# B&R Automation Studio project Tmp_Explorer_V1
Automation Studio 4.12.7.113 SP; technology packages: mappView 5.24.4

## Configuration Simulation

CPU PC_any, AutomationRuntime B4.53, Build 4.1.2, Vc V4.52.0

### Task classes (Cpu.sw)
```
Cyclic#8 (cycle 10000 us):
  FileExplor <- mappFileExplorer.FileExplorer.prg
  NETdevice <- mappFileExplorer.NETdevice.prg
  USBdevice <- mappFileExplorer.USBdevice.prg
Binaries: TCData, mvLoader, udbdef, ashwac, Role, ashwd, arconfig, iomap, OpcUaMap, asfw, sysconf, User
Libraries: standard, asieccon, astime, runtime, fileio, asbrstr, asusb
```

### Hardware
```
PC : PC_any v1.1.0.0 (OrderNumber=PC)
  ConfigurationID = Tmp_Explorer_V1_Simulation
  Cyclic8Duration = 10000
  FileDevice1
  FileDeviceName1 = USER
  FileDevicePath1 = C:\Temp
  FileDevice2
  FileDeviceName2 = SYSTEM
  FileDevicePath2 = C:\projects
  ActivateOpcUa = 1
  OpcUaInformationModels_PV_Version = 1
```

## Configuration X20CPU

CPU X20CP1583, AutomationRuntime B4.53, Build 4.1.2, Vc V4.52.0

CPU X20CP3585, AutomationRuntime J4.93, Build 4.1.2, Safety 0.0, Vc V4.52.0

### Task classes (Cpu.sw)
```
Cyclic#8:
  FileExplor <- mappFileExplorer.FileExplorer.prg
  UsbDevice <- USBdevice.UsbDevice.prg
  NetDevice <- NETdevice.NetDevice.prg
Binaries: udbdef, mvLoader, TCData, OpcUaMap, arconfig, User, Role, iomap, asfw, ashwac, ashwd, sysconf
Libraries: FileIO, runtime, AsBrStr, AsUSB, standard, IecCheck, sys_lib, AsHttp, AsMem, AsARCfg, AsZip, astime, asieccon, AsICMP
```

### Task classes (Cpu.sw)
```
Cyclic#8:
  USBdevice <- mappFileExplorer.USBdevice.prg
  FileExplor <- mappFileExplorer.FileExplorer.prg
Libraries: FileIO, runtime, AsBrStr, AsUSB, standard
```

### Hardware
```
X20CP3585 : X20CP3585 v1.10.0.0
  Connector IF2:
    ActivateDevice = 1
  Connector IF3:
    DNAConfiguration = manual
  ConfigurationID = Tmp_Explorer_V1_Config1
  UserPartitionSize = 200
  Simulation = 1
  VolatileGlobalPvSize = 200000
  FileDevice1
  FileDeviceName1 = USER
  FileDevicePath1 = F:\
  FileDevice2
  FileDeviceName2 = SYSTEM
  FileDevicePath2 = C:\
  FtpUser1
  FtpUsername1 = br
  FtpUserPassword1 = B9fKGuUbjkGCgEptWUpgQ1eJbLeEvMYqPBCteWUIcCw=
  FtpUserSalt1 = wEo/3/qm
  FTPAccessRight1 = 0
  ActivateOpcUa = 1
  OpcUaInformationModels_PV_Version = 1
```

## Logical view

Binary libraries used (declarations not repeated): operator, runtime, astime, AsIecCon, FileIO, AsBrStr, AsUSB, standard, sys_lib, AsHttp, AsMem, AsARCfg, AsZip, AsICMP

### Package Logical/Libraries - Global libraries

### Library Logical/Libraries/IecCheck (IEC)
Depends on: sys_lib, AsBrStr

#### IecCheck.st - Implementation file
```iecst
(* Check divisor for SINT division *)
FUNCTION CheckDivSint
	IF divisor=0 THEN
		CheckDivSint:=1;
		MakeEntry(55555,divisor,'CheckDivSint');
	ELSE
		CheckDivSint:=divisor;
	END_IF
END_FUNCTION

(* Check divisor for USINT division *)
FUNCTION CheckDivUsint
	IF divisor=0 THEN
		CheckDivUsint:=1;
		MakeEntry(55555,divisor,'CheckDivUsint');
	ELSE
		CheckDivUsint:=divisor;
	END_IF
END_FUNCTION

(* Check divisor for INT division *)
FUNCTION CheckDivInt
	IF divisor=0 THEN
		CheckDivInt:=1;
		MakeEntry(55555,divisor,'CheckDivInt');
	ELSE
		CheckDivInt:=divisor;
	END_IF
END_FUNCTION

(* Check divisor for UINT division *)
FUNCTION CheckDivUint
	IF divisor=0 THEN
		CheckDivUint:=1;
		MakeEntry(55555,divisor,'CheckDivUint');
	ELSE
		CheckDivUint:=divisor;
	END_IF
END_FUNCTION

(* Check divisor for DINT division *)
FUNCTION CheckDivDint
	IF divisor=0 THEN
		CheckDivDint:=1;
		MakeEntry(55555,divisor,'CheckDivDint');
	ELSE
		CheckDivDint:=divisor;
	END_IF
END_FUNCTION

(* Check divisor for UDINT division *)
FUNCTION CheckDivUdint
	IF divisor=0 THEN
		CheckDivUdint:=1;
		MakeEntry(55555,divisor,'CheckDivUdint');
	ELSE
		CheckDivUdint:=divisor;
	END_IF
END_FUNCTION

(* Check divisor for REAL division *)
FUNCTION CheckDivReal
	IF divisor=0 THEN
		CheckDivReal:=1;
		MakeEntry(55555,0,'CheckDivReal');
	ELSE
		CheckDivReal:=divisor;
	END_IF
END_FUNCTION

(* Check divisor for LREAL division *)
FUNCTION CheckDivLReal
	IF divisor=0 THEN
		CheckDivLReal:=1;
		MakeEntry(55555,0,'CheckDivLReal');
	ELSE
		CheckDivLReal:=divisor;
	END_IF
END_FUNCTION

(* Check range for array access *)
FUNCTION CheckBounds
	IF index < lower THEN
		CheckBounds := lower;
		MakeEntry(55555,index,'CheckBounds');
	ELSIF index > upper THEN
		CheckBounds := upper;
		MakeEntry(55555,index,'CheckBounds');
	ELSE
		CheckBounds := index;
	END_IF
END_FUNCTION

(* Check range for enumeration *)
FUNCTION CheckRange
	IF value < lower THEN
		CheckRange := lower;
		MakeEntry(55555,value,'CheckRange');
	ELSIF value > upper THEN
		CheckRange := upper;
		MakeEntry(55555,value,'CheckRange');
	ELSE
		CheckRange := value;
	END_IF
END_FUNCTION

(* Check range for subrange of signed data types *)
FUNCTION CheckSignedSubrange
	IF value < lower THEN
		CheckSignedSubrange := lower;
		MakeEntry(55555,value,'CheckSignedSubrange');
	ELSIF value > upper THEN
		CheckSignedSubrange := upper;
		MakeEntry(55555,value,'CheckSignedSubrange');
	ELSE
		CheckSignedSubrange := value;
	END_IF
END_FUNCTION

(* Check range for subrange of unsigned data types *)
FUNCTION CheckUnsignedSubrange
	IF value < lower THEN
		CheckUnsignedSubrange := lower;
		MakeEntry(55555,value,'CheckUnsignedSubrange');
	ELSIF value > upper THEN
		CheckUnsignedSubrange := upper;
		MakeEntry(55555,value,'CheckUnsignedSubrange');
	ELSE
		CheckUnsignedSubrange := value;
	END_IF
END_FUNCTION

(* Check address when reading dynamic variables *)
FUNCTION CheckReadAccess
	IF address=0 THEN
		(* TODO: Insert an appropriate code, see AutomationStudio help for further information *)
		MakeEntry(55555,address,'Read from NULL');
	END_IF

	CheckReadAccess:=0;
END_FUNCTION

(* Check address when writing dynamic variables *)
FUNCTION CheckWriteAccess
	IF address=0 THEN
		(* TODO: Insert an appropriate code, see AutomationStudio help for further information *)
		MakeEntry(55555,address,'Write to NULL');
	END_IF

	CheckWriteAccess:=0;
END_FUNCTION

(* Makes an entry (log book entry) in the error log book *)
FUNCTION MakeEntry
		status_name := ST_name(0,ADR(taskname),ADR(group));

		brsstrcpy(ADR(out_text),ADR(text));
		brsstrcat(ADR(out_text),ADR(' > in task > '));
  		brsstrcat(ADR(out_text),ADR(taskname));
		MakeEntry := ADR(out_text);
		ERRxfatal(number,index,ADR(out_text));
END_FUNCTION
```

- Visualisation Logical/mappView (not shown)

### ExplorerTypes.typ
```iecst
TYPE
	ClientInfoType : 	STRUCT
		userId : WSTRING[80];
		isValid : BOOL;
		ipAddress : WSTRING[15];
		languageId : WSTRING[2];
		screenResolution : WSTRING[32];
		slotId : SINT;
	END_STRUCT;
	expSTATE :
		( (*Explorer state machine*)
		EXP_WAIT,
		EXP_READ_DIR,
		EXP_READ_DIR_1,
		EXP_READ_DIR_2,
		EXP_READ_DIR_3,
		EXP_READ_DIR_4,
		EXP_DIR_CHANGE,
		EXP_COPY_ALL,
		EXP_FILE_COPY,
		EXP_FILE_DELETE,
		EXP_FILE_RENAME,
		EXP_FILE_VIEW,
		EXP_FILE_DOWNLOAD,
		EXP_FILE_DOWNLOAD_1,
		EXP_FILE_DOWNLOAD_2,
		EXP_FILE_DOWNLOAD_3,
		EXP_FILE_DOWNLOAD_4,
		EXP_FILE_DOWNLOAD_5,
		EXP_FILE_DOWNLOAD_DIR,
		EXP_FILE_UPLOAD,
		EXP_FILE_UPLOAD_1,
		EXP_FILE_UPLOAD_2,
		EXP_FILE_UPLOAD_3,
		EXP_FILE_UPLOAD_4,
		EXP_DIR_COPY,
		EXP_DIR_CREATE,
		EXP_DIR_DELETE,
		EXP_DIR_RENAME,
		EXP_OVERWRITE_1,
		EXP_OVERWRITE_2
		);
	expERR : 	STRUCT  (*Sub structure error*)
		text : STRING[150]; (* Error text *)
		state : expSTATE; (* Error step *)
	END_STRUCT;
	expCMD : 	STRUCT  (*Sub structure commands*)
		refresh : BOOL; (*Read directory and file names from devices *)
		dir_change : BOOL; (*Change current directory *)
		dir_create : BOOL; (*Create a new directory *)
		copy : BOOL; (*Copy selected item from device a TO device b *)
		copy_all : BOOL; (*Copy all items from device a TO device b	*)
		view_file : BOOL; (*View selected file in mappView*)
		delete : BOOL; (*Delete selected file *)
		rename : BOOL; (*Rename selected file*)
		download : BOOL; (*Download selected file*)
		upload : BOOL; (*Upload file to target*)
	END_STRUCT;
	expPAR : 	STRUCT  (*Sub structure parameters*)
		device_active : STRING[40]; (*Active device name *)
		device_list : ARRAY[0..6]OF STRING[40]; (*List of all devices*)
		item_filter : STRING[EXPL_ITEM_LENGTH]; (*Only show files with this extension	*)
		new_name : STRING[EXPL_ITEM_LENGTH]; (*Name for for directory create and rename*)
		dir_path : STRING[EXPL_DIR_PATH_LENGTH]; (*Current directory path	*)
	END_STRUCT;
	expDAT : 	STRUCT  (*Sub structure data*)
		item_list : ARRAY[0..EXPL_LIST_NUM]OF STRING[EXPL_ITEM_LENGTH]; (*List with file names	*)
		item_size : ARRAY[0..EXPL_LIST_NUM]OF STRING[EXPL_SIZE_LENGTH]; (*List with file sizes*)
		item_num : UINT; (*Number of files	 displayed*)
		device_free : UINT; (*Free memory on device in MB*)
		device_size : UINT; (*Total memory size of device in MB*)
	END_STRUCT;
	expVIS : 	STRUCT  (*Sub structure visualization*)
		item_selected : UINT; (*Current selected file *)
		enable_button_set_1 : BOOL; (*Enable or disable buttons copy and delete*)
		enable_button_set_2 : BOOL; (*Enable or disable buttons refresh and create*)
		view_file_path : STRING[EXPL_DIR_PATH_LENGTH]; (*Full path for viewing file*)
		view_file : BOOL; (*Show message box on error*)
		download_file_url : STRING[200]; (*File upload and download url*)
		upload_overwrite_request : BOOL; (*Show message box to overwrite file*)
		upload_overwrite_response : USINT; (*Response from message box overwrite file*)
		reload_upload : BOOL; (*Reload upload button*)
		double_click_event : USINT; (*Helper variable for double click in item list*)
		device_list : ARRAY[0..6]OF STRING[80]; (* Device name *)
	END_STRUCT;
	expMAIN : 	STRUCT  (*Main explorer structure*)
		CMD : ARRAY[0..1]OF expCMD; (* Command structure *)
		PAR : ARRAY[0..1]OF expPAR; (* Parameter structure *)
		DAT : ARRAY[0..1]OF expDAT; (*Data structure*)
		VIS : ARRAY[0..1]OF expVIS; (*Visualization structure*)
		ERR : expERR; (* Error structure *)
		status_no : UINT; (*Shows the status as number*)
		status_text : STRING[50]; (*Shows the status as text*)
	END_STRUCT;
END_TYPE
```

### ExplorerVariables.var
```iecst
VAR CONSTANT
	EXPL_DIR_PATH_LENGTH : UINT := 200; (*Maximum length for the complete path *)
	EXPL_LIST_NUM : UINT := 100; (*Maximum number if files and folders that can be listed *)
	EXPL_ITEM_LENGTH : USINT := 50; (*Maximum length for a file or folder name *)
	EXPL_SIZE_LENGTH : USINT := 15; (*Maximum length for a file or folder size*)
	EXPL_UPLOAD_DOWNLOAD_SIZE : UDINT := 5000000; (*Maximum size of memory allocated for uploading and downloading files*)
	EXPL_DEVICE_LIST : ARRAY[0..6] OF STRING[40] := ['USER','SYSTEM','USB_DEVICE1','USB_DEVICE2','USB_DEVICE3','NET_DEVICE','']; (*List of predefined devices *)
END_VAR
VAR
	EXPL_VIEW_FILTER : ARRAY[0..9] OF STRING[5] := ['csv','xml','txt','bmp','jpg',5('')]; (*Files extensions than can be used with the view command*)
	EXPL : expMAIN; (*Explorer main structure*)
END_VAR
```

### Program Logical/mappFileExplorer/FileExplorer (ANSIC)

#### Main.c - Init, cyclic, exit code
```c
	//******************************** B&R * Application TB-West *******************************************
	//	Function:	Mini explorer
	//	Autor:		S.Stricker
	//  Version:	1.00
	//	Changed:	03.09.2019
	//	Error numbers:
	//	50000		Selected item name is empty
	//	50001		This is not a valid item name
	//	50010		Device is not defined
	//	50011		Item list is not defined
	//	50012		Maximum entry parameter is 0
	//	50100		Maximum number of files reached
	//	50200		File name exceeds maximum length
	//	50201		Directory name exceeds maximum length
	//	50202		Directory path exceeds maximum length
	//	50203		Directory path critical error
	//******************************************************************************************************

#include <bur/plctypes.h>

#ifdef _DEFAULT_INCLUDES
	#include <AsDefault.h>
#endif

void CreateError(UINT nr, USINT SIDE, STRING txt[100], typMain_EXP *EXPL);
void WorkingStatus(typMain_EXP *EXPL, UDINT str);
void CreateCompletePath(STRING path[DIR_PATH_SIZE+MAX_ITEM_SIZE], STRING target[MAX_ITEM_SIZE], UDINT return_path);
void InsertRecName(typMain_EXP *EXPL, STRING new_name[DIR_PATH_SIZE], STRING size[15], UINT SIDE);
void SelectItem(typMain_EXP *EXPL, USINT SOURCE);
BOOL IsInstr(STRING string1[MAX_ITEM_SIZE], STRING string2[MAX_ITEM_SIZE]);

//******************************************************************************************************
// Init Part
//******************************************************************************************************
void _INIT ProgramInit(void)
{
	brsmemcpy((UDINT)EXPL.PAR[0].device_list, (UDINT)DEVICE_LIST, sizeof(DEVICE_LIST));
	brsmemcpy((UDINT)EXPL.PAR[1].device_list, (UDINT)DEVICE_LIST, sizeof(DEVICE_LIST));
	brsstrcpy((UDINT)EXPL.PAR[0].device_active, (UDINT)EXPL.PAR[0].device_list[0]);
	brsstrcpy((UDINT)EXPL.PAR[1].device_active, (UDINT)EXPL.PAR[1].device_list[0]);
}

//******************************************************************************************************
// Cyclic Part
//******************************************************************************************************
void _CYCLIC ProgramCyclic(void)
{
	USINT SIDE;
	SIDE = side;

	//--------------------------------------------------------------------------------------------------
	// Check if parameters are valid
	if (brsstrcmp((UDINT)EXPL.PAR[SIDE].device_active, (UDINT)"") == 0)
	{
		CreateError(50010, SIDE, "device is not defined", &EXPL);
		return;
	}
	if(brsstrlen((UDINT)EXPL.PAR[SIDE].dir_path) >= DIR_PATH_SIZE)
	{
		CreateError(50203, SIDE, "Directory path critical error", &EXPL);
		return;
	}
	// ------------------------------------------------------------------------------------------------
	// Track filter change
	if((FILTER_AUTO_REFRESH) && (brsstrcmp((UDINT)old_filter[SIDE], (UDINT)EXPL.PAR[SIDE].item_filter) != 0))
	{
		brsstrcpy((UDINT)old_filter[SIDE], (UDINT)EXPL.PAR[SIDE].item_filter);
		EXPL.CMD[SIDE].refresh	= 1;
	}

	// ------------------------------------------------------------------------------------------------
	// Track device name change
	if(brsstrcmp((UDINT)device_active_old[SIDE], (UDINT)EXPL.PAR[SIDE].device_active) != 0)
	{
		brsstrcpy((UDINT)EXPL.PAR[SIDE].dir_path, (UDINT)"");
		EXPL.CMD[SIDE].refresh	= 1;
	}
	brsstrcpy((UDINT)device_active_old[SIDE], (UDINT)EXPL.PAR[SIDE].device_active);

	// ------------------------------------------------------------------------------------------------
	// Set switches for HMI
	if(EXPL.DAT[SIDE].item_num > 0) EXPL.VIS[SIDE].enable_copy_delete = 1;
	else EXPL.VIS[SIDE].enable_copy_delete = 0;

	// ------------------------------------------------------------------------------------------------
	// Generate device name list
	brsmemset((UDINT)EXPL.VIS[SIDE].device_list, 0, sizeof(EXPL.VIS[SIDE].device_list));
	for (x = 0; x < sizeof(EXPL.VIS[SIDE].device_list)/sizeof(EXPL.VIS[SIDE].device_list[0]); x++)
	{
		if (brsstrcmp((UDINT)EXPL.PAR[SIDE].device_list[x], (UDINT)"") != 0)
		{
			brsstrcpy((UDINT)EXPL.VIS[SIDE].device_list[x], (UDINT)"{\"value\":\"");
			brsstrcat((UDINT)EXPL.VIS[SIDE].device_list[x], (UDINT)EXPL.PAR[SIDE].device_list[x]);
			brsstrcat((UDINT)EXPL.VIS[SIDE].device_list[x], (UDINT)"\",\"text\":\"");
			brsstrcat((UDINT)EXPL.VIS[SIDE].device_list[x], (UDINT)EXPL.PAR[SIDE].device_list[x]);
			brsstrcat((UDINT)EXPL.VIS[SIDE].device_list[x], (UDINT)"\"}");
		}
	}

	// ------------------------------------------------------------------------------------------------
	// Handle double click for directory change
	if(EXPL.VIS[SIDE].double_click_dir_change > 0)
	{
		DoubleClickDirChange.PT = 50;
		DoubleClickDirChange.IN = 1;
		TON_10ms(&DoubleClickDirChange);
		if(EXPL.VIS[SIDE].double_click_dir_change > 1)
		{
			DoubleClickDirChange.IN = 0;
			TON_10ms(&DoubleClickDirChange);
			EXPL.VIS[SIDE].double_click_dir_change = 0;
			if(brsmemcmp((UDINT)EXPL.DAT[SIDE].item_list[EXPL.VIS[SIDE].item_selected], (UDINT)"(DIR)", 5) == 0 ||
			   brsmemcmp((UDINT)EXPL.DAT[SIDE].item_list[EXPL.VIS[SIDE].item_selected], (UDINT)"..", 2) == 0) EXPL.CMD[SIDE].dir_change = 1;
		}
	}
	if(DoubleClickDirChange.Q)
	{
		DoubleClickDirChange.IN = 0;
		TON_10ms(&DoubleClickDirChange);
		if(EXPL.VIS[SIDE].double_click_dir_change > 0) EXPL.VIS[SIDE].double_click_dir_change = EXPL.VIS[SIDE].double_click_dir_change - 1;
	}

	for (cycles = 0; cycles < override; cycles++)
	{
		// ------------------------------------------------------------------------------------------------
		// Break if no command is set
		if (EXPL.CMD[SIDE].refresh 		== 0 &&
			EXPL.CMD[SIDE].dir_change	== 0 &&
			EXPL.CMD[SIDE].dir_create 	== 0 &&
			EXPL.CMD[SIDE].copy 		== 0 &&
			EXPL.CMD[SIDE].copyall 		== 0 &&
			EXPL.CMD[SIDE].delete 		== 0)
		{
			// --------------------------------------------------------------------------------------------
			// Show current state
			brsstrcpy((UDINT)EXPL.status, (UDINT)"Waiting...");
			// --------------------------------------------------------------------------------------------
			// If selection is out of range set it to maximum
			if ((EXPL.VIS[SIDE].item_selected > EXPL.DAT[SIDE].item_num - 1) &&
				(EXPL.DAT[SIDE].item_num != 0)) EXPL.VIS[SIDE].item_selected = EXPL.DAT[SIDE].item_num - 1;
			side = !side;
			// Enable buttons when command is active
			EXPL.VIS[0].enable_refresh_create = 1;
			EXPL.VIS[1].enable_refresh_create = 1;
			break;
		}
		// Disable buttons when command is active
		EXPL.VIS[0].enable_copy_delete = 0;
		EXPL.VIS[1].enable_copy_delete = 0;
		EXPL.VIS[0].enable_refresh_create = 0;
		EXPL.VIS[1].enable_refresh_create = 0;
		//**************************************************************************************************
		// Cyclic Part
		//**************************************************************************************************
		switch (step)
		{
			//**********************************************************************************************
			// Wait for command
			//**********************************************************************************************
			case STP_WAIT:
				// ----------------------------------------------------------------------------------------
				// Command refresh
				if (EXPL.CMD[SIDE].refresh == 1) step = STP_READ_DIR;
				// ----------------------------------------------------------------------------------------
				// Command directory change
				if (EXPL.CMD[SIDE].dir_change == 1)
				{
					// ------------------------------------------------------------------------------------
					// Check if directory name is empty
					if (brsstrcmp((UDINT)EXPL.DAT[SIDE].item_list[EXPL.VIS[SIDE].item_selected], (UDINT)"") == 0)	CreateError(50000, SIDE, "directory name is empty", &EXPL);
						// Check if directory name is valid
					else if((brsmemcmp((UDINT)EXPL.DAT[SIDE].item_list[EXPL.VIS[SIDE].item_selected], (UDINT)"(DIR)", 5) != 0) && (brsmemcmp((UDINT)EXPL.DAT[SIDE].item_list[EXPL.VIS[SIDE].item_selected], (UDINT)"..", 2) != 0)) CreateError(50001, SIDE, "this is not a valid directory name", &EXPL);
						// Check if new directory name fits into string
					else if(brsstrlen((UDINT)EXPL.DAT[SIDE].item_list[EXPL.VIS[SIDE].item_selected]) - 5 + brsstrlen((UDINT)EXPL.PAR[SIDE].dir_path) + 1 >= DIR_PATH_SIZE) CreateError(50202, SIDE, "directory path exceeds maximum length", &EXPL);
					else step = STP_DIR_CHANGE;
				}
				// ----------------------------------------------------------------------------------------
				// Command directory create
				if (EXPL.CMD[SIDE].dir_create == 1)
				{
					// ------------------------------------------------------------------------------------
					// Check if new directory name is empty
					if (brsstrcmp((UDINT)EXPL.PAR[SIDE].dir_name, (UDINT)"") == 0) CreateError(50000, SIDE, "directory name is empty", &EXPL);
						// Check if new directory name fits into path string
					else if(brsstrlen((UDINT)EXPL.PAR[SIDE].dir_name) + brsstrlen((UDINT)EXPL.PAR[SIDE].dir_path) + 1 >= DIR_PATH_SIZE) CreateError(50202, SIDE, "directory path name exceeds maximum length", &EXPL);
						// Check if new directory name fits into directory name string
					else if(brsstrlen((UDINT)EXPL.PAR[SIDE].dir_name) + 5 >= MAX_ITEM_SIZE) CreateError(50201, SIDE, "directory name exceeds maximum length", &EXPL);
					else step = STP_DIR_CREATE;
				}
				// ----------------------------------------------------------------------------------------
				// Command copy
				if (EXPL.CMD[SIDE].copy == 1)
				{
					// ------------------------------------------------------------------------------------
					// Make sure that user chooses a valid item
					if (brsstrcmp((UDINT)EXPL.DAT[SIDE].item_list[EXPL.VIS[SIDE].item_selected], (UDINT)"..") == 0)			CreateError(50001, SIDE, "this is not a valid item name", &EXPL);
					else if(brsmemcmp((UDINT)EXPL.DAT[SIDE].item_list[EXPL.VIS[SIDE].item_selected], (UDINT)"(DIR)", 5) == 0)	step = STP_DIR_COPY;
					else																														step = STP_FILE_COPY;
				}
				// ----------------------------------------------------------------------------------------
				// Command copy all
				if (EXPL.CMD[SIDE].copyall == 1) step = STP_COPY_ALL;
				// ----------------------------------------------------------------------------------------
				// Command delete
				if (EXPL.CMD[SIDE].delete == 1)
				{
					// ------------------------------------------------------------------------------------
					// Check if directory name is empty
					if (brsstrcmp((UDINT)EXPL.DAT[SIDE].item_list[EXPL.VIS[SIDE].item_selected], (UDINT)"") == 0)	CreateError(50000, SIDE, "item name is empty", &EXPL);
						// Check if new directory name fits into string
					else if(brsstrlen((UDINT)EXPL.DAT[SIDE].item_list[EXPL.VIS[SIDE].item_selected]) + brsstrlen((UDINT)EXPL.PAR[SIDE].dir_path) + 1 >= DIR_PATH_SIZE + MAX_ITEM_SIZE) CreateError(50202, SIDE, "directory path exceeds maximum length", &EXPL);
						// Make sure that user chooses a valid item
					else if(brsstrcmp((UDINT)EXPL.DAT[SIDE].item_list[EXPL.VIS[SIDE].item_selected], (UDINT)"..") == 0) CreateError(50001, SIDE, "this is not a valid item name", &EXPL);
						// Delete a directory
					else if(brsmemcmp((UDINT)EXPL.DAT[SIDE].item_list[EXPL.VIS[SIDE].item_selected], (UDINT)"(DIR)", 5) == 0)	step = STP_DIR_DELETE;
						// Delete a file
					else																											step = STP_FILE_DELETE;
				}
				// ----------------------------------------------------------------------------------------
				// Clear errors
				if (EXPL.CMD[SIDE].refresh 		== 1 ||
					EXPL.CMD[SIDE].copy 		== 1 ||
					EXPL.CMD[SIDE].copyall 		== 1 ||
					EXPL.CMD[SIDE].dir_create 	== 1 ||
					EXPL.CMD[SIDE].delete		== 1)
				{
					brsstrcpy((UDINT)EXPL.ERR.txt, (UDINT)"");
					EXPL.ERR.nr   		= 0;
					EXPL.ERR.step 		= 0;
				}
				break;
			//**********************************************************************************************
			// Read directory information
			//**********************************************************************************************
			case STP_READ_DIR:
				// Show current state
				WorkingStatus(&EXPL, (UDINT)"read directory...");
				// ----------------------------------------------------------------------------------------
				// Clear all entrys
				brsmemset((UDINT)&EXPL.DAT[SIDE], 0, sizeof(EXPL.DAT[SIDE]));
				EXPL.VIS[SIDE].item_selected = 0;
				EXPL.DAT[SIDE].item_num = 0;
				// ----------------------------------------------------------------------------------------
				// Add .. for directory up
				if((brsstrcmp((UDINT)EXPL.PAR[SIDE].dir_path, (UDINT)"\\") != 0) &&
				   (brsstrcmp((UDINT)EXPL.PAR[SIDE].dir_path, (UDINT)"") != 0))
				{
					brsstrcpy((UDINT)EXPL.DAT[SIDE].item_list, (UDINT)"..");
					EXPL.DAT[SIDE].item_num = 1;
				}
				// ----------------------------------------------------------------------------------------
				// Set values and get device dir
				DInfo.enable 	= 1;
				DInfo.pDevice	= (UDINT)EXPL.PAR[SIDE].device_active;
				DInfo.pPath 	= (UDINT)EXPL.PAR[SIDE].dir_path;
				DirInfo(&DInfo);

				// ----------------------------------------------------------------------------------------
				// ->Success
				if (DInfo.status == OK) step = STP_READ_DIR_1;
				// ----------------------------------------------------------------------------------------
				// Device is not available
				else if (DInfo.status == fiERR_FILE_DEVICE )
				{
					brsstrcpy((UDINT)EXPL.DAT[SIDE].item_list, (UDINT)"not connected");
					CreateError(DInfo.status, SIDE, "not connected", &EXPL);
				}
				// ----------------------------------------------------------------------------------------
				// Device is not available
				else if (DInfo.status == fiERR_DEVICE_MANAGER )
				{
					brsstrcpy((UDINT)EXPL.DAT[SIDE].item_list, (UDINT)"not connected");
					CreateError(DInfo.status, SIDE, "check device name and path", &EXPL);
				}
				else if (DInfo.status != 65535) CreateError(DInfo.status, SIDE, "error dir info", &EXPL);
				break;
			//**********************************************************************************************
			// Open directory
			//**********************************************************************************************
			case STP_READ_DIR_1:
				// ----------------------------------------------------------------------------------------
				// Set values and get device dir
				DOpen.enable 	= 1;
				DOpen.pDevice	= (UDINT)EXPL.PAR[SIDE].device_active;
				DOpen.pName 	= (UDINT)EXPL.PAR[SIDE].dir_path;
				DirOpen(&DOpen);

				// ----------------------------------------------------------------------------------------
				// ->Success
				if (DOpen.status == OK) step	= STP_READ_DIR_2;
				else if (DOpen.status != 65535) CreateError(DOpen.status, SIDE, "error dir open", &EXPL);
				break;
			//**********************************************************************************************
			// Read file directory information
			//**********************************************************************************************
			case STP_READ_DIR_2:
				// ----------------------------------------------------------------------------------------
				// Initialize read directory structure
				DRead.enable 	= 1;
				DRead.ident		= DOpen.ident;
				DRead.pData 	= (UDINT)&lDirReadData;
				DRead.data_len 	= sizeof(lDirReadData);
				DirReadEx(&DRead);

				// ----------------------------------------------------------------------------------------
				// ->Success
				if (DRead.status == OK)
				{
					// ------------------------------------------------------------------------------------
					// Verify that we still have space in list
					if (EXPL.DAT[SIDE].item_num < sizeof(EXPL.DAT[SIDE].item_list)/sizeof(EXPL.DAT[SIDE].item_list[0]))
					{
						// --------------------------------------------------------------------------------
						// Verify that extension is equal to filter
						if ((brsstrlen((UDINT)EXPL.PAR[SIDE].item_filter) == 0) || (IsInstr((STRING*)lDirReadData.Filename, EXPL.PAR[SIDE].item_filter)))
						{
							// ----------------------------------------------------------------------------
							// Read file information
							if (lDirReadData.Mode == fiFILE)
							{
								if (brsstrlen((UDINT)lDirReadData.Filename) < MAX_ITEM_SIZE-5)
								{
									brsmemset((UDINT)tmp_str1, 0, sizeof(tmp_str1));
									brsmemcpy((UDINT)tmp_str1, (UDINT)lDirReadData.Filename, brsstrlen((UDINT)lDirReadData.Filename));
									// --------------------------------------------------------------------
									// Append file size
									if(lDirReadData.Filelength > 999999)
									{
										brsitoa((lDirReadData.Filelength/1000000), (UDINT)tmp_str2);
										brsstrcat((UDINT)tmp_str2, (UDINT)"M");
									}
									else if(lDirReadData.Filelength > 999)
									{
										brsitoa((lDirReadData.Filelength/1000), (UDINT)tmp_str2);
										brsstrcat((UDINT)tmp_str2, (UDINT)"K");
									}
									else
									{
										brsitoa((lDirReadData.Filelength), (UDINT)tmp_str2);
									}
									brsmemcpy((UDINT)tmp_str1 + MAX_ITEM_SIZE - brsstrlen((UDINT)tmp_str2) - 1, (UDINT)tmp_str2, brsstrlen((UDINT)tmp_str2));
									InsertRecName(&EXPL, tmp_str1, tmp_str2, SIDE);
									EXPL.DAT[SIDE].item_num++;
								}
								else CreateError(50200, SIDE, "file name exceeds maximum length", &EXPL);
							}
							// ----------------------------------------------------------------------------
							// Read directory information
							else if((brsstrcmp((UDINT)lDirReadData.Filename, (UDINT)".")  != 0) &&
								    (brsstrcmp((UDINT)lDirReadData.Filename, (UDINT)"..") != 0) &&
									(brsstrcmp((UDINT)lDirReadData.Filename, (UDINT)"System Volume Information") != 0))
								{
								if (brsstrlen((UDINT)lDirReadData.Filename) < MAX_ITEM_SIZE-5)
								{
									// Copy directory name
									brsstrcpy((UDINT)tmp_str1, (UDINT)"(DIR)");
									brsstrcat((UDINT)tmp_str1, (UDINT)lDirReadData.Filename);
									InsertRecName(&EXPL, tmp_str1, "", SIDE);
									EXPL.DAT[SIDE].item_num++;
								}
								else CreateError(50201, SIDE, "directory name exceeds maximum length", &EXPL);
							}
						}
					}
					else CreateError(50100, SIDE, "maximum number of files reached", &EXPL);
				}
				else if (DRead.status == fiERR_NO_MORE_ENTRIES) step = STP_READ_DIR_3;
					// ----------------------------------------------------------------------------------------
				else if (DRead.status != 65535) CreateError(DRead.status, SIDE, "error dir read", &EXPL);
				break;
			//**********************************************************************************************
			// Close directory information
			//**********************************************************************************************
			case STP_READ_DIR_3:
				// ----------------------------------------------------------------------------------------
				// Initialize read directory structure
				DClose.enable 	= 1;
				DClose.ident	= DOpen.ident;
				DirClose(&DClose);

				// ----------------------------------------------------------------------------------------
				// ->Success
				if (DClose.status == OK)
				{
					// Select item after copy->refresh
					if(do_select != 0)	SelectItem(&EXPL, do_select-1);
					do_select = 0;
					// Reset command and return to wait state
					EXPL.CMD[SIDE].refresh	= 0;
					DClose.ident			= 0;
					step					= STP_WAIT;
				}
					// ----------------------------------------------------------------------------------------
				else if (DClose.status != 65535) CreateError(DClose.status, SIDE, "error dir close", &EXPL);
				break;
			//**********************************************************************************************
			// Change directory
			//**********************************************************************************************
			case STP_DIR_CHANGE:
				// ----------------------------------------------------------------------------------------
				// Move one directory up
				if(brsstrcmp((UDINT)EXPL.DAT[SIDE].item_list[EXPL.VIS[SIDE].item_selected], (UDINT)"..") == 0)
				{
					x = brsstrlen((UDINT)EXPL.PAR[SIDE].dir_path);
					while(x>0)
					{
					if(brsmemcmp((UDINT)(UDINT)(EXPL.PAR[SIDE].dir_path + x), (UDINT)"/", 1) == 0) break;
					else brsmemset((UDINT)(UDINT)(EXPL.PAR[SIDE].dir_path + x), 0, 1);
					x--;
					}
					brsmemset((UDINT)(UDINT)(EXPL.PAR[SIDE].dir_path + x), 0, 1);
				}
					// ----------------------------------------------------------------------------------------
					// Move one directory down
				else
				{
					brsstrcat((UDINT)EXPL.PAR[SIDE].dir_path, (UDINT)"/");
					brsstrcat((UDINT)EXPL.PAR[SIDE].dir_path, (UDINT)EXPL.DAT[SIDE].item_list[EXPL.VIS[SIDE].item_selected] + 5);
					EXPL.CMD[SIDE].refresh = 1;
				}
				// Reset command and return to wait state
				EXPL.VIS[SIDE].item_selected	= 0;
				EXPL.CMD[SIDE].dir_change 		= 0;
				EXPL.CMD[SIDE].refresh 			= 1;
				step							= STP_WAIT;
				break;
			//**********************************************************************************************
			// Copy all items
			//**********************************************************************************************
			case STP_COPY_ALL:
				// Show current state
				WorkingStatus(&EXPL, (UDINT)"copying files...");

				EXPL.VIS[SIDE].item_selected = 0;
				// ----------------------------------------------------------------------------------------
				// Skip dots at list beginning
				if (brsstrcmp((UDINT)EXPL.DAT[SIDE].item_list[EXPL.VIS[SIDE].item_selected], (UDINT)"..") == 0)		EXPL.VIS[SIDE].item_selected++;
				// Check first entry
				if(brsmemcmp((UDINT)EXPL.DAT[SIDE].item_list[EXPL.VIS[SIDE].item_selected], (UDINT)"(DIR)", 5) == 0)	step = STP_DIR_COPY;
				else																													step = STP_FILE_COPY;
				break;
			//**********************************************************************************************
			// Copy files
			//**********************************************************************************************
			case STP_FILE_COPY:
				// Show current state
				WorkingStatus(&EXPL, (UDINT)"copying file...");

				// -----------------------------------------------------------------.----------------------
				// Proceed with copy all until last file is copied
				if ((EXPL.VIS[SIDE].item_selected < sizeof(EXPL.DAT[SIDE].item_list)/sizeof(EXPL.DAT[SIDE].item_list[0])) && (EXPL.VIS[SIDE].item_selected < EXPL.DAT[SIDE].item_num))
				{
					// ------------------------------------------------------------------------------------
					// Check if file name is empty
					if (brsstrcmp((UDINT)EXPL.DAT[SIDE].item_list[EXPL.VIS[SIDE].item_selected], (UDINT)"") != 0)
					{
						// --------------------------------------------------------------------------------
						// Check if new file name fits into string
						if(brsstrlen((UDINT)EXPL.DAT[SIDE].item_list[EXPL.VIS[SIDE].item_selected]) < MAX_ITEM_SIZE)
						{
							// ----------------------------------------------------------------------------
							// Initialize copy structure
							CreateCompletePath((void*)EXPL.PAR[SIDE].dir_path, (void*)EXPL.DAT[SIDE].item_list[EXPL.VIS[SIDE].item_selected], (UDINT)&tmp_str3);
							CreateCompletePath((void*)EXPL.PAR[!SIDE].dir_path, (void*)EXPL.DAT[SIDE].item_list[EXPL.VIS[SIDE].item_selected], (UDINT)&tmp_str4);
							FCopy.enable 	= 1;
							FCopy.pSrcDev	= (UDINT)EXPL.PAR[SIDE].device_active;
							FCopy.pSrc		= (UDINT)&tmp_str3;
							FCopy.pDestDev  = (UDINT)EXPL.PAR[!SIDE].device_active;
							FCopy.pDest		= (UDINT)&tmp_str4;
							FCopy.option 	= FILE_OW_DETMEM;
							FileCopy(&FCopy);

							// ----------------------------------------------------------------------------
							// ->Success
							if ((FCopy.status == OK) && (EXPL.CMD[SIDE].copy == 1))
							{
								// Select entry, reset command and refresh directory
								if(COPY_AUTO_REFRESH) EXPL.CMD[!SIDE].refresh = 1;
								if(COPY_AUTO_SELECT) do_select = SIDE + 1;
								EXPL.CMD[SIDE].copy	= 0;
								step = STP_WAIT;
							}
							// ----------------------------------------------------------------------------
							// Proceed with next file
							else if (FCopy.status == OK) EXPL.VIS[SIDE].item_selected++;
							else if (FCopy.status != 65535)	CreateError(FCopy.status, SIDE, "error copying file", &EXPL);
						}
						else CreateError(50200, SIDE, "file name exceeds maximum length", &EXPL);
					}
					else CreateError(50000, SIDE, "file name is empty", &EXPL);
				}
				// ----------------------------------------------------------------------------------------
				// Finish copy all
				else
				{
					// Reset command and refresh directory
					if(COPY_AUTO_REFRESH) EXPL.CMD[!SIDE].refresh = 1;
					EXPL.CMD[SIDE].copyall			= 0;
					EXPL.VIS[SIDE].item_selected 	= 0;
					step				= STP_WAIT;
				}
				break;
			//**********************************************************************************************
			// Copy directory
			//**********************************************************************************************
			case STP_DIR_COPY:
				// Show current state
				WorkingStatus(&EXPL, (UDINT)"copying directory...");

				// ----------------------------------------------------------------------------------------
				// Proceed with copy all until last file is copied
				if ((EXPL.VIS[SIDE].item_selected < sizeof(EXPL.DAT[SIDE].item_list)/sizeof(EXPL.DAT[SIDE].item_list[0])) && (EXPL.VIS[SIDE].item_selected < EXPL.DAT[SIDE].item_num))
				{
					if (brsstrcmp((UDINT)EXPL.DAT[SIDE].item_list[EXPL.VIS[SIDE].item_selected], (UDINT)"") != 0)
					{
					// --------------------------------------------------------------------------------
					// Check if new directory name fits into path string
					if(brsstrlen((UDINT)EXPL.DAT[SIDE].item_list[EXPL.VIS[SIDE].item_selected]) + brsstrlen((UDINT)EXPL.PAR[!SIDE].dir_path) + 1 < DIR_PATH_SIZE)
					{
					// ----------------------------------------------------------------------------
					// Initialize copy structure
					CreateCompletePath((void*)EXPL.PAR[SIDE].dir_path, (void*)EXPL.DAT[SIDE].item_list[EXPL.VIS[SIDE].item_selected], (UDINT)&tmp_str3);
					CreateCompletePath((void*)EXPL.PAR[!SIDE].dir_path, (void*)EXPL.DAT[SIDE].item_list[EXPL.VIS[SIDE].item_selected], (UDINT)&tmp_str4);
					DCopy.enable 	= 1;
					DCopy.pSrcDev	= (UDINT)EXPL.PAR[SIDE].device_active;
					DCopy.pSrcDir	= (UDINT)&tmp_str3;
					DCopy.pDestDev 	= (UDINT)EXPL.PAR[!SIDE].device_active;
					DCopy.pDestDir 	= (UDINT)&tmp_str4;
					DCopy.option 	= fiOVERWRITE;
					DirCopy(&DCopy);

					// ----------------------------------------------------------------------------
					// ->Success
					if ((DCopy.status == OK) && (EXPL.CMD[SIDE].copy == 1))
					{
					// Reset command and refresh directory
					if(COPY_AUTO_REFRESH) 	EXPL.CMD[!SIDE].refresh = 1;
					if(COPY_AUTO_SELECT) 	do_select = SIDE + 1;
					EXPL.CMD[SIDE].copy	= 0;
					step		= STP_WAIT;
					}
					// ----------------------------------------------------------------------------
					// Proceed with next directory
					else if (DCopy.status == OK)
					{
					EXPL.VIS[SIDE].item_selected++;
					// Switch to file copy when no more directory can be found
					if(brsmemcmp((UDINT)EXPL.DAT[SIDE].item_list[EXPL.VIS[SIDE].item_selected], (UDINT)"(DIR)", 5) != 0)	step = STP_FILE_COPY;
					}
					else if (DCopy.status != 65535) CreateError(DCopy.status, SIDE, "error copying directory", &EXPL);
					}
					else CreateError(50202, SIDE, "directory path name exceeds maximum length", &EXPL);
					}
					else CreateError(50000, SIDE, "directory name is empty", &EXPL);
				}
					// ----------------------------------------------------------------------------------------
					// Finish copy all
				else
				{
					// Reset command and refresh directory
					if(COPY_AUTO_REFRESH) EXPL.CMD[!SIDE].refresh = 1;
					EXPL.CMD[SIDE].copyall			= 0;
					EXPL.VIS[SIDE].item_selected 	= 0;
					step				= STP_WAIT;
				}
				break;
			//**********************************************************************************************
			// Delete selected file
			//**********************************************************************************************
			case STP_FILE_DELETE:
				// Show current state
				WorkingStatus(&EXPL, (UDINT)"deleting file...");

				// ----------------------------------------------------------------------------------------
				// Initialize file delete structure
				CreateCompletePath((void*)EXPL.PAR[SIDE].dir_path, (void*)EXPL.DAT[SIDE].item_list[EXPL.VIS[SIDE].item_selected], (UDINT)&tmp_str3);
				FDelete.enable		= 1;
				FDelete.pDevice 	= (UDINT)EXPL.PAR[SIDE].device_active;
				FDelete.pName		= (UDINT)tmp_str3;
				FileDelete(&FDelete);

				// ----------------------------------------------------------------------------------------
				// ->Success
				if (FDelete.status == OK)
				{
					// Reset command and return to wait state
					EXPL.CMD[SIDE].delete 	= 0;
					EXPL.CMD[SIDE].refresh  = 1;
					step = STP_WAIT;
				}
				else if (FDelete.status != 65535) CreateError(FDelete.status, SIDE, "error deleting file", &EXPL);
				break;
			//**********************************************************************************************
			// Create new directory
			//**********************************************************************************************
			case STP_DIR_CREATE:
				// Show current state
				WorkingStatus(&EXPL, (UDINT)"creating directory...");

				// ----------------------------------------------------------------------------------------
				// Initialize directory create structure
				CreateCompletePath((void*)EXPL.PAR[SIDE].dir_path, (void*)EXPL.PAR[SIDE].dir_name, (UDINT)&tmp_str3);
				DCreate.enable	= 1;
				DCreate.pDevice = (UDINT)EXPL.PAR[SIDE].device_active;
				DCreate.pName 	= (UDINT)&tmp_str3;
				DirCreate(&DCreate);

				// ----------------------------------------------------------------------------------------
				// ->Success
				if (DCreate.status == OK)
				{
					// Reset command and return to wait state
					EXPL.CMD[SIDE].dir_create 	= 0;
					EXPL.CMD[SIDE].refresh 		= 1;
					step = STP_WAIT;
				}
				else if (DCreate.status != 65535) CreateError(DCreate.status, SIDE, "error creating directory", &EXPL);
				break;
			//**********************************************************************************************
			// Delete selected directory
			//**********************************************************************************************
			case STP_DIR_DELETE:
				// Show current state
				WorkingStatus(&EXPL, (UDINT)"deleting directory...");

				// ----------------------------------------------------------------------------------------
				// Initialize directory delete structure
				CreateCompletePath((void*)EXPL.PAR[SIDE].dir_path, (void*)EXPL.DAT[SIDE].item_list[EXPL.VIS[SIDE].item_selected], (UDINT)&tmp_str3);
				DDelete.enable	= 1;
				DDelete.pDevice = (UDINT)EXPL.PAR[SIDE].device_active;
				DDelete.pName 	= (UDINT)&tmp_str3;
				DirDeleteEx(&DDelete);

				// ----------------------------------------------------------------------------------------
				// ->Success
				if (DDelete.status == OK)
				{
					// Reset command and return to wait state
					EXPL.CMD[SIDE].delete 	= 0;
					EXPL.CMD[SIDE].refresh = 1;
					step		= STP_WAIT;
				}
				else if (DDelete.status != 65535) CreateError(DDelete.status, SIDE, "error deleting directory", &EXPL);
				break;
		}
	}
}

//******************************************************************************************************
// Create complete path string
//******************************************************************************************************
void CreateCompletePath(STRING path[DIR_PATH_SIZE+MAX_ITEM_SIZE], STRING target[MAX_ITEM_SIZE], UDINT return_path)
{
	STRING 	tmp[MAX_ITEM_SIZE];
	brsmemset((UDINT)&tmp, 0, MAX_ITEM_SIZE);
	brsstrcpy((UDINT)return_path, (UDINT)path);
	// ------------------------------------------------------------------------------------------------
	// Filter directory name
	if(brsmemcmp((UDINT)target, (UDINT)"(DIR)", 5) == 0)
		brsmemcpy((UDINT)tmp, (UDINT)(target+5), brsstrlen((UDINT)target)-5);
	else
		brsstrcpy((UDINT)tmp, (UDINT)target);

	// ------------------------------------------------------------------------------------------------
	// Create directory path
	brsstrcat((UDINT)return_path, (UDINT)"/");
	brsstrcat((UDINT)return_path, (UDINT)tmp);
}

//******************************************************************************************************
// Raise error function
//******************************************************************************************************
void CreateError(UINT nr, USINT SIDE, STRING txt[100], typMain_EXP *EXPL)
{
	if (nr == fiERR_NOT_ENOUGH_FREEMEM) brsstrcpy((UDINT)EXPL->ERR.txt, (UDINT)"not enough memory available on the target device");
	else if (nr == fiERR_FILE_DEVICE) 	brsstrcpy((UDINT)EXPL->ERR.txt, (UDINT)"device is not connected");
	else if (nr == fiERR_INVALID_PATH) 	brsstrcpy((UDINT)EXPL->ERR.txt, (UDINT)"directory is too long or has invalid characters");
	else if (nr == fiERR_DIR_NOT_EXIST) brsstrcpy((UDINT)EXPL->ERR.txt, (UDINT)"directory path dont exist");
	else brsstrcpy((UDINT)EXPL->ERR.txt, (UDINT)txt);
	// Convert to error structure
	if (SIDE == 0) 	brsstrcat((UDINT)EXPL->ERR.txt, (UDINT)" on side a");
	else			brsstrcat((UDINT)EXPL->ERR.txt, (UDINT)" on side b");
	EXPL->ERR.nr   	= nr;
	EXPL->ERR.step 	= step;
	// Reset all commands
	brsmemset((UDINT)&EXPL->CMD[SIDE], 0, sizeof(EXPL->CMD[SIDE]));
	brsmemset((UDINT)&EXPL->CMD[!SIDE], 0, sizeof(EXPL->CMD[!SIDE]));
	if (DClose.ident == 0) 	step = STP_WAIT;
	else					step = STP_READ_DIR_3;
}

//******************************************************************************************************
// Working status
//******************************************************************************************************
void WorkingStatus(typMain_EXP *EXPL, UDINT str)
{
	animation++;
	if (animation == 80) animation = 0;
	brsmemset((UDINT)EXPL->status, 0, sizeof(EXPL->status));
	brsstrcpy((UDINT)EXPL->status, (UDINT)str);
	switch(animation)
	{
		case 0 ... 19	: brsstrcat((UDINT)EXPL->status, (UDINT)"/"); break;
		case 20 ... 39	: brsstrcat((UDINT)EXPL->status, (UDINT)"-"); break;
		case 40 ... 59	: brsstrcat((UDINT)EXPL->status, (UDINT)"\\"); break;
		case 60 ... 79	: brsstrcat((UDINT)EXPL->status, (UDINT)"|"); break;
	}
}

//******************************************************************************************************
// Fill new folder or directory name
//******************************************************************************************************
void InsertRecName(typMain_EXP *EXPL, STRING new_name[MAX_ITEM_SIZE], STRING size[15], UINT SIDE)
{
	DINT 				lx		= 0;
	DINT 				ly		= 0;
	DINT  				lSort	= 0;

	// Set up start values for iteration
	if (EXPL->DAT[SIDE].item_num != 0) ly = EXPL->DAT[SIDE].item_num - 1;
	lx = ly;
	// Start itteration	search
	while (ly > 1)
	{
		// Check current entry
		lSort = brsstrcmp((UDINT)new_name, (UDINT)EXPL->DAT[SIDE].item_list[ly]);
		// Solve new search range
		if (ly % 2 == 0) 	ly = ly / 2;
		else				ly = ly / 2 + 1;
		// New range is lower or higher than current
		if (lSort > 0)
		{
			lx = lx + ly;
			if (lx > EXPL->DAT[SIDE].item_num) lx = EXPL->DAT[SIDE].item_num;
		}
		else
		{
			lx = lx - ly;
			if (lx < 1) lx = 1;
		}
	}
	// New entry is this, next or previous
	lSort = brsstrcmp((UDINT)new_name, (UDINT)EXPL->DAT[SIDE].item_list[lx]);
	if ((lSort > 0) && (lx != EXPL->DAT[SIDE].item_num)) lx++;
	else if (lx > 0)
	{
		lSort = brsstrcmp((UDINT)new_name, (UDINT)EXPL->DAT[SIDE].item_list[lx-1]);
		if (lSort < 0) lx--;
	}
	// Force ".." at beginning of list
	if ((lx == 0) && (brsstrcmp((UDINT)"..", (UDINT)EXPL->DAT[SIDE].item_list)) == 0) lx++;
	// Move all data entrys backwards and fill in new entry
	brsmemmove((UDINT)EXPL->DAT[SIDE].item_list[lx+1],(UDINT)EXPL->DAT[SIDE].item_list[lx], (EXPL->DAT[SIDE].item_num - lx) * (MAX_ITEM_SIZE + 1));
	brsstrcpy((UDINT)EXPL->DAT[SIDE].item_list[lx], (UDINT)new_name);

	// Create data structure for vis size listbox
	brsmemmove((UDINT)EXPL->DAT[SIDE].item_size[lx+1],(UDINT)EXPL->DAT[SIDE].item_size[lx], (EXPL->DAT[SIDE].item_num - lx) * (15 + 1));
	brsstrcpy((UDINT)EXPL->DAT[SIDE].item_size[lx], (UDINT)size);
}

//******************************************************************************************************
// Select item
//******************************************************************************************************
void SelectItem(typMain_EXP *EXPL, USINT SOURCE)
{
	UINT x = 0;

	for(x=0;x<EXPL->DAT[!SOURCE].item_num;x++) if(brsstrcmp((UDINT)EXPL->DAT[SOURCE].item_list[EXPL->VIS[SOURCE].item_selected], (UDINT)EXPL->DAT[!SOURCE].item_list[x]) == 0) break;
	EXPL->VIS[!SOURCE].item_selected = x;
}

//******************************************************************************************************
// Is second string in first string
//******************************************************************************************************
BOOL IsInstr(STRING string1[MAX_ITEM_SIZE], STRING string2[MAX_ITEM_SIZE])
{
	UINT x = 0;

	if(brsstrlen((UDINT)string1)>brsstrlen((UDINT)string2))
	{
		for(x=0;x<=brsstrlen((UDINT)string1)-brsstrlen((UDINT)string2);x++) if(brsmemcmp((UDINT)string1 + x, (UDINT)string2, brsstrlen((UDINT)string2)) == 0) return 1;
	}
	return 0;
}
```

#### Types.typ - Local data types
```iecst
TYPE
	STEP :
		(
		STP_WAIT,
		STP_READ_DIR,
		STP_READ_DIR_1,
		STP_READ_DIR_2,
		STP_READ_DIR_3,
		STP_DIR_CHANGE,
		STP_COPY_ALL,
		STP_FILE_COPY,
		STP_FILE_DELETE,
		STP_DIR_COPY,
		STP_DIR_CREATE,
		STP_DIR_DELETE
		);
END_TYPE
```

#### Variables.var - Local variables
```iecst
(*Local constants*)
VAR CONSTANT
	OK : USINT := 0; (*Status OK *)
	FILTER_AUTO_REFRESH : BOOL := TRUE; (*Auto refresh when filter changes *)
	COPY_AUTO_SELECT : USINT := 1; (*Select target item after copying *)
	COPY_AUTO_REFRESH : USINT := 1; (*Refresh items after copying *)
END_VAR
(*Local Variables*)
VAR
	side : BOOL := FALSE; (*Current side *)
	step : expSTATE := (0); (*Main step index *)
	animation : USINT := 0; (*Animation for working status	*)
	do_select : USINT := 0; (*Select item after copying *)
	old_filter : ARRAY[0..1] OF STRING[EXPL_ITEM_LENGTH]; (*Track filter change *)
	has_oversized_items : BOOL;
	tmp_str1 : STRING[EXPL_DIR_PATH_LENGTH]; (* Temporary STRING variable *)
	tmp_str2 : STRING[EXPL_DIR_PATH_LENGTH]; (* Temporary STRING variable *)
	tmp_str3 : STRING[EXPL_DIR_PATH_LENGTH]; (* Temporary STRING variable *)
	tmp_str4 : STRING[EXPL_DIR_PATH_LENGTH]; (* Temporary STRING variable *)
	lx : UDINT := 0; (* Index	*)
	ly : UINT;
	double_click_timer : TON_10ms;
	device_active_old : ARRAY[0..1] OF STRING[40];
	response_header : httpResponseHeader_t;
	response_header_data : STRING[300];
	download_timeout : TON_10ms;
	upload_delay : TON_10ms;
	upload_response : ARRAY[0..1] OF STRING[1000];
	file_name_start : DINT;
	file_name_len : DINT;
	file_data_start : DINT;
	file_data_len : DINT;
	dir_path : STRING[EXPL_DIR_PATH_LENGTH];
	device_active : STRING[40];
	item_name : STRING[EXPL_DIR_PATH_LENGTH];
END_VAR
(*Local function calls*)
VAR
	DInfo : DirInfo;
	DOpen : DirOpen;
	DRead : DirReadEx;
	DClose : DirClose;
	FWrite : FileWrite;
	FCreate : FileCreate;
	FOpen : FileOpen;
	FRead : FileReadEx;
	FClose : FileClose;
	FCopy : FileCopy;
	FDelete : FileDelete;
	FRename : FileRename;
	DCopy : DirCopy;
	DCreate : DirCreate;
	DDelete : DirDeleteEx;
	DRename : DirRename;
	DMemInfo : DevMemInfo;
	DevLink_0 : DevLink;
	lDirReadData : fiDIR_READ_EX_DATA;
	AsMemPartCreate_0 : AsMemPartCreate;
	AsMemPartAllocClear_0 : AsMemPartAllocClear;
	WebServiceUpload : ARRAY[0..1] OF httpService := [2((0))];
	WebserviceDownload : httpService := (0);
	zipArchive_0 : zipArchive;
END_VAR
(*Local constants*)
VAR CONSTANT
	YES : USINT := 1;
	NO : USINT := 2;
	SKIP : USINT := 3;
	ERR_EMPTY_ITEM : UINT := 50000; (*Selected item name is empty	*)
	ERR_INVALID_ITEM_NAME : UINT := 50001; (*This is not a valid item name*)
	ERR_DEVICE_UNDEFINED : UINT := 50010; (*Device is not defined*)
	ERR_MAX_FILES_REACHED : UINT := 50100; (*Maximum number of files reached*)
	ERR_NAME_EXCEEDS_MAX : UINT := 50200; (*File name exceeds maximum length*)
	ERR_DIR_EXCEEDS_MAX : UINT := 50201; (*Directory name exceeds maximum length*)
	ERR_PATH_EXCEEDS_MAX : UINT := 50202; (*Directory path exceeds maximum length*)
	ERR_PATH_CRITICAL : UINT := 50203; (*Directory path critical error*)
	ERR_PATH_RECURSIVE : UINT := 50204; (*Can not copy directory into itself*)
	ERR_MEM_ALLOC : UINT := 50300; (*Memory allocation for file upload and download failed*)
	ERR_MEM_DOWNLOAD : UINT := 50310; (*Size of download file exceeds maximum*)
	ERR_TIMEOUT_DOWNLOAD : UINT := 50320; (*Download response timed out*)
	ERR_DIR_DOWNLOAD_INVALID : UINT := 50331; (*This is not a valid directory for downloading*)
	ERR_POS_NAME_UPLOAD : UINT := 50400; (*Can not find filename in upload response*)
	ERR_SIZE_NAME_UPLOAD : UINT := 50401; (*Can not determine end of filename in upload response*)
	ERR_LEN_NAME_UPLOAD : UINT := 50402; (*Filename is too long in upload response*)
	ERR_POS_DATA_UPLOAD : UINT := 50403; (*Can not find data in upload response*)
	ERR_SIZE_DATA_UPLOAD : UINT := 50404; (*Can not determine end of data in upload response*)
	ERR_MEM_UPLOAD : UINT := 50410; (*Size of upload file exceeds maximum size*)
END_VAR
```

#### LocalFunctions.fun - not listed in the package file held
```iecst
FUNCTION ReplaceString : BOOL
	VAR_INPUT
		dataSTR : UDINT;
		searchSTR : UDINT;
		replaceSTR : UDINT;
		first : BOOL;
	END_VAR
	VAR
		idx : UDINT;
	END_VAR
END_FUNCTION

FUNCTION IsInstr : BOOL
	VAR_INPUT
		string1 : UDINT;
		string2 : UDINT;
	END_VAR
	VAR
		idx : UDINT;
	END_VAR
END_FUNCTION

FUNCTION FindInMem : DINT
	VAR_INPUT
		data1 : UDINT;
		len1 : UDINT;
		data2 : UDINT;
		len2 : UDINT;
		direction : BOOL;
	END_VAR
	VAR
		idx : UDINT;
	END_VAR
END_FUNCTION

{REDUND_ERROR} FUNCTION CreateError : expSTATE (*TODO: Add your comment here*) (*$GROUP=User,$CAT=User,$GROUPICON=User.png,$CATICON=User.png*)
	VAR_INPUT
		nr : UINT;
		side : BOOL;
		step : expSTATE;
		text : STRING[150];
		EXPL : REFERENCE TO expMAIN;
	END_VAR
END_FUNCTION

FUNCTION InsertRecName : BOOL
	VAR_INPUT
		EXPL : REFERENCE TO expMAIN;
		new_name : STRING[EXPL_ITEM_LENGTH];
		size : STRING[15];
		side : BOOL;
	END_VAR
	VAR
		idx : DINT;
		idy : DINT;
		lSort : DINT;
	END_VAR
END_FUNCTION

FUNCTION WorkingStatus : USINT
	VAR_INPUT
		EXPL : REFERENCE TO expMAIN;
		str : UDINT;
		animation : USINT;
	END_VAR
END_FUNCTION

FUNCTION CreateCompletePath : BOOL
	VAR_INPUT
		path : STRING[EXPL_DIR_PATH_LENGTH];
		target : STRING[EXPL_ITEM_LENGTH];
		return_path : UDINT;
	END_VAR
	VAR
		tmp : STRING[EXPL_ITEM_LENGTH];
	END_VAR
END_FUNCTION

FUNCTION String2DataProvider : BOOL
	VAR_INPUT
		SourceString : UDINT;
		TargetString : UDINT;
	END_VAR
END_FUNCTION
```

#### LocalFunctions.st - not listed in the package file held
```iecst
//******************************************************************************************************
// Create mappView data provider string
//******************************************************************************************************
FUNCTION String2DataProvider
	brsstrcpy(TargetString, ADR('{"value":"'));
	brsstrcat(TargetString, SourceString);
	brsstrcat(TargetString, ADR('","text":"'));
	brsstrcat(TargetString, SourceString);
	brsstrcat(TargetString, ADR('"}'));
	String2DataProvider := TRUE;
END_FUNCTION

//******************************************************************************************************
// Raise error function
//******************************************************************************************************
FUNCTION CreateError
	// Generate for known errors
	IF (nr = fiERR_NOT_ENOUGH_FREEMEM) THEN
		EXPL.ERR.text := 'not enough memory available on the target device';
	ELSIF (nr = fiERR_FILE_DEVICE) THEN
		EXPL.ERR.text := 'device is not connected';
	ELSIF (nr = fiERR_INVALID_PATH) THEN
		EXPL.ERR.text := 'directory is too long, does not exist or has invalid characters';
	ELSIF (nr = fiERR_DIR_NOT_EXIST) THEN
		EXPL.ERR.text := 'directory does not exist';
	ELSIF (nr = fiERR_FILE_DEVICE) THEN
		EXPL.ERR.text := 'directory path does not exist';
	ELSIF (nr = fiERR_DIR_ALREADY_EXIST) THEN
		EXPL.ERR.text := 'directory or file already exists';
	ELSIF (nr = fiERR_EXIST) THEN
		EXPL.ERR.text := 'error uploading file already exists';
	ELSE
		EXPL.ERR.text := text;
	END_IF
	// Convert to error structure
	IF (side = 0) THEN
		brsstrcat(ADR(EXPL.ERR.text), ADR(' on side a'));
	ELSE
		brsstrcat(ADR(EXPL.ERR.text), ADR(' on side b'));
	END_IF
	EXPL.status_no 	:= nr;
	EXPL.ERR.state 	:= step;
	// When error occurs in dir read call dir close before reporting error
	IF (step = EXP_READ_DIR_2) THEN
		CreateError := EXP_READ_DIR_3;
	// When error occurs in file write call file close before reporting error
	ELSIF(step = EXP_FILE_UPLOAD_2) THEN
		CreateError := EXP_FILE_UPLOAD_3;
	ELSE
		// Reset all commands
		brsmemset(ADR(EXPL.CMD[side]), 0, SIZEOF(EXPL.CMD[side]));
		brsmemset(ADR(EXPL.CMD[NOT side]), 0, SIZEOF(EXPL.CMD[NOT side]));
		CreateError := EXP_WAIT;
	END_IF
END_FUNCTION

//******************************************************************************************************
// Create complete path string
//******************************************************************************************************
FUNCTION CreateCompletePath
	brsmemset(ADR(tmp), 0, EXPL_ITEM_LENGTH);
	brsstrcpy(return_path, ADR(path));

	// ------------------------------------------------------------------------------------------------
	// Filter directory name
	IF(brsmemcmp(ADR(target), ADR('(DIR)'), 5) = 0) THEN
		brsmemcpy(ADR(tmp), ADR(target)+5, brsstrlen(ADR(target))-5);
	ELSE
		brsstrcpy(ADR(tmp), ADR(target));
	END_IF

	// ------------------------------------------------------------------------------------------------
	// Create directory path
	IF(path <> '/') THEN
		brsstrcat(return_path, ADR('/'));
	END_IF
	brsstrcat(return_path, ADR(tmp));
	//	brsstrcat(return_path, ADR('/'));

	CreateCompletePath := FALSE;
END_FUNCTION

//******************************************************************************************************
// Working status
//******************************************************************************************************
FUNCTION WorkingStatus
	animation := animation+1;

	IF (animation = 80) THEN
		animation := 0;
	END_IF

	brsmemset(ADR(EXPL.status_text), 0, SIZEOF(EXPL.status_text));
	brsstrcpy(ADR(EXPL.status_text), str);
	CASE(animation) OF
		0..19	: brsstrcat(ADR(EXPL.status_text), ADR('/'));
		20..39	: brsstrcat(ADR(EXPL.status_text), ADR('-'));
		40..59	: brsstrcat(ADR(EXPL.status_text), ADR('\'));
		60..79	: brsstrcat(ADR(EXPL.status_text), ADR('|'));
	END_CASE;
	WorkingStatus := animation;
END_FUNCTION

//******************************************************************************************************
// Fill new folder or directory name
//******************************************************************************************************
FUNCTION InsertRecName
	// Set up start values for iteration
	IF (EXPL.DAT[side].item_num <> 0) THEN
		idy := EXPL.DAT[side].item_num - 1;
	END_IF
	idx := idy;

	// Start iteration	search
	WHILE (idy > 1) DO
		// Check current entry
		lSort := brsstrcmp(ADR(new_name), ADR(EXPL.DAT[side].item_list[idy]));
		// Solve new search range
		IF (idy MOD 2 = 0) THEN
			idy := idy / 2;
		ELSE
			idy := idy / 2 + 1;
		END_IF
		// New range is lower or higher than current
		IF (lSort > 0) THEN
			idx := idx + idy;
			IF (idx > UINT_TO_INT(EXPL.DAT[side].item_num)) THEN
				idx := EXPL.DAT[side].item_num;
			END_IF
		ELSE
			idx := idx - idy;
			IF (idx < 1) THEN
				idx := 1;
			END_IF
		END_IF
	END_WHILE;

	// New entry is this, next or previous
	lSort := brsstrcmp(ADR(new_name), ADR(EXPL.DAT[side].item_list[idx]));
	IF (lSort > 0 AND idx <> UINT_TO_INT(EXPL.DAT[side].item_num)) THEN
		idx := idx +1;
	ELSIF (idx > 0) THEN
		lSort := brsstrcmp(ADR(new_name), ADR(EXPL.DAT[side].item_list[idx-1]));
		IF (lSort < 0) THEN
			idx := idx - 1;
		END_IF
	END_IF

	// Force ".." at beginning of list
	IF (idx = 0 AND EXPL.DAT[side].item_list[0] = '..') THEN
		idx := idx + 1;
	END_IF
	// Move all data entrys backwards and fill in new entry
	IF(idx < EXPL_LIST_NUM) THEN
		brsmemmove(ADR(EXPL.DAT[side].item_list[idx+1]),ADR(EXPL.DAT[side].item_list[idx]), (EXPL.DAT[side].item_num - idx) * SIZEOF(EXPL.DAT[side].item_list[0]));
		brsmemmove(ADR(EXPL.DAT[side].item_size[idx+1]),ADR(EXPL.DAT[side].item_size[idx]), (EXPL.DAT[side].item_num - idx) * SIZEOF(EXPL.DAT[side].item_size[0]));
	END_IF
	brsstrcpy(ADR(EXPL.DAT[side].item_list[idx]), ADR(new_name));
	// Create data structure for vis size list
	brsstrcpy(ADR(EXPL.DAT[side].item_size[idx]), ADR(size));

	InsertRecName := TRUE;
END_FUNCTION

//******************************************************************************************************
// Is second string in first string
//******************************************************************************************************
FUNCTION IsInstr
	IF (brsstrlen(string1) > brsstrlen(string2)) THEN
		FOR idx:=0 TO brsstrlen(string1) - brsstrlen(string2) DO
			IF (brsmemcmp(string1 + idx, string2, brsstrlen(string2)) = 0) THEN
				IsInstr := TRUE;
				EXIT;
			END_IF
		END_FOR;
	END_IF
END_FUNCTION

//******************************************************************************************************
// Find second data in first data
//******************************************************************************************************
FUNCTION FindInMem
	FindInMem := -1;
	IF (len1 > len2) THEN
		IF(direction) THEN
			idx := len1 - len2;
			WHILE(idx > 0) DO
				IF (brsmemcmp(data1 + idx, data2, len2) = 0) THEN
					FindInMem := idx;
					EXIT;
				END_IF
				idx := idx - 1;
			END_WHILE;
		ELSE
			FOR idx:=0 TO len1 - len2 DO
				IF (brsmemcmp(data1 + idx, data2, len2) = 0) THEN
					FindInMem := idx;
					EXIT;
				END_IF
			END_FOR;
		END_IF
	END_IF
END_FUNCTION

//******************************************************************************************************
// Find and replace string
//******************************************************************************************************
FUNCTION ReplaceString
	IF (brsstrlen(dataSTR) >= brsstrlen(searchSTR)) THEN
		FOR idx:=0 TO brsstrlen(dataSTR) - brsstrlen(searchSTR) DO
			IF (brsmemcmp(dataSTR + idx, searchSTR, brsstrlen(searchSTR)) = 0) THEN
				// Move data around
				brsmemmove(dataSTR + idx + brsstrlen(replaceSTR), dataSTR + idx + brsstrlen(searchSTR), brsstrlen(dataSTR) - brsstrlen(searchSTR) + 1);
				brsmemcpy(dataSTR + idx, replaceSTR, brsstrlen(replaceSTR));
				// Set found flag and exit if only one hit is needed
				ReplaceString := TRUE;
				IF(first) THEN
					EXIT;
				END_IF
				// Correct index for next search
				IF(brsstrlen(replaceSTR) > 0) THEN
					idx := idx + brsstrlen(replaceSTR);
				END_IF
				idx := idx - 1;
				// Exit if no data is left
				IF (brsstrlen(dataSTR) = 0 OR brsstrlen(dataSTR) < brsstrlen(searchSTR)) THEN
					EXIT;
				END_IF
			END_IF
		END_FOR;
	END_IF
END_FUNCTION
```
